# EPICS autosave request: isegHVPSU/isegHVPSU_settings.req
$(P):DISABLE
$(P):SET_I1_TRIP.A
$(P):SET_I1_TRIP.B
$(P):SET_I1_TRIP.C
$(P):SET_I1_TRIP.D
$(P):SET_I1_TRIP_DEMAND
$(P):SET_I2_TRIP.A
$(P):SET_I2_TRIP.B
$(P):SET_I2_TRIP.C
$(P):SET_I2_TRIP.D
$(P):SET_I2_TRIP_DEMAND
$(P):SET_V1_DEMAND
$(P):SET_V1_RAMP_DEMAND
$(P):SET_V1_RAMP_RATE.A
$(P):SET_V1_RAMP_RATE.B
$(P):SET_V1_RAMP_RATE.C
$(P):SET_V1_SET.A
$(P):SET_V1_SET.B
$(P):SET_V1_SET.C
$(P):SET_V1_SET.D
$(P):SET_V2_DEMAND
$(P):SET_V2_RAMP_DEMAND
$(P):SET_V2_RAMP_RATE.A
$(P):SET_V2_RAMP_RATE.B
$(P):SET_V2_RAMP_RATE.C
$(P):SET_V2_SET.A
$(P):SET_V2_SET.B
$(P):SET_V2_SET.C
$(P):SET_V2_SET.D
